# B&R Automation Studio project AsProject
Automation Studio 6.5.2.12; Starter Automation Studio project.; technology packages: mappConnect 6.1.0, mappView 6.6.0, OpcUaCs 6.5.0, OpcUaFx 6.6.0

## Configuration StarterConfig

CPU 5PC900.TS17-04, AutomationRuntime 6.5.1, Build 11.3.0

### Task classes (Cpu.sw)
```
Cyclic#1 (cycle 2000 us, tolerance 0 us):
  test <- test.prg
  TestTypes <- TestTypes.prg
  demo <- demo.prg
  demoGlobal <- demoGlobal.prg
  Page <- Page.prg
Binaries: udbdef, TCData, FWRules, mvLoader, mvDatApi, mvConfig, ashwd, ashwac, User, sysconf, asfw, arconfig, iomap, UaCsConfig, Config, BRRole, Role
Libraries: UaCore, ArSsl, FileIO, runtime
```

### Hardware
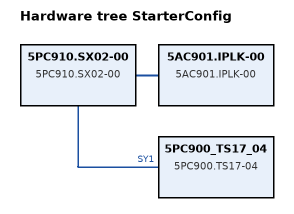
```
5AC901.IPLK-00 : 5AC901.IPLK-00 v2.1.0.0  [SS -> 5PC910.SX02-00.SS2]
  Connector IF1:
    DNAConfiguration = manual
5PC900_TS17_04 : 5PC900.TS17-04 v2.2.0.0  [SY -> 5PC910.SX02-00.SY1]
  ConfigurationID = Starter_StarterConfig
  UserPartitionSize = 300
  Simulation = 1
  UserRamDevice = PCI.2.IPLK.SRAM
  UserRamSize = 500000
  RemMemDevice = PCI.2.IPLK.SRAM
  RemMemSize = 120000
  PermanentPvSize = 10000
  RemanentGlobalPvSize = 105000
  VolatileGlobalPvSize = 1000000
  TimerDeviceType = EPLX2X
  TimerDevice = 5AC901.IPLK-00.IF1
  IdleTaskClass = 3
  TaskClassIdleTime = 8000
  Cyclic1Duration = 2000
  Cyclic1Tolerance = 0
  Cyclic2Duration = 10000
  Cyclic3Duration = 20000
  Cyclic3Tolerance = 40000
  FileDevice1
  FileDeviceName1 = USER
  FileDevicePath1 = USER_PATH
  TimeZone = 25
  ActivateFtpServer = 1
  FtpUser1
  FtpUsername1 = dev
  FtpUserPassword1 = NYwXHzz4INzZvtlFBMOTmjZqrH4JRkY3Uye1yrmlNSg=  // dev
  FtpUserSalt1 = s9/ksXy4
  FTPAccessRight1 = 0
  FTPdevice1 = ALL
  ActivateWebServer = 1
  ActivateSdm = 1
  SdmColor = colorRGB
  ActivateHypervisor = 1
5PC910.SX02-00 : 5PC910.SX02-00 v2.1.2.0
  Connector IF1:
    AssignedOperatingSystem = ARemb
  Connector IF3:
    AssignedOperatingSystem = ARemb
    ActivateDevice = 1
  Connector IF4:
    AssignedOperatingSystem = ARemb
    ActivateDevice = 1
  Connector IF10:
    OperatingSystem = ARemb
    ActivateDevice = 1
  Connector IF5:
    AssignedOperatingSystem = ARemb
  Connector IF6:
    AssignedOperatingSystem = ARemb
  Connector IF7:
    AssignedOperatingSystem = ARemb
  Connector IF8:
    AssignedOperatingSystem = ARemb
  Connector IF9:
    AssignedOperatingSystem = ARemb
```

### BRRole.brrole - 5PC900_TS17_04/AccessAndSecurity/UserRoleSystem/BRRole.brrole
```
Element BR_Anonymous (Type=BRRole)
Element BR_Engineer (Type=BRRole)
Element BR_Observer (Type=BRRole)
Element BR_SafetyAdmin (Type=BRRole)
Element BR_SecurityAdmin (Type=BRRole)
```

- Physical/StarterConfig/5PC900_TS17_04/IoMap.iom: same as Physical/StarterConfig/5PC900_TS17_04/Cpu.per
- Physical/StarterConfig/5PC900_TS17_04/PvMap.vvm: same as Physical/StarterConfig/5PC900_TS17_04/Cpu.per
### Config.mappconnect - 5PC900_TS17_04/mappConnect/Config.mappconnect
```
Element mapp Connect Configuration (Type=mappconnect)
  WebServerProtocol:
    WebServerPortSsl = 8443
    Interface = All
    SSLConfiguration = 
  WebServerEndpointConfiguration:
    Endpoint[1]:
      Endpoint = /Index.html
      Roles
    Endpoint[2]:
      Endpoint = /api/*
      Roles
    Endpoint[3]:
      Endpoint = /*
      Roles
  OpcUaServerWhitelist:
    OpcUaServer[1]:
      Url = opc.tcp://127.0.0.1:4840
```

## Logical view

### Global.var - Global variables
```iecst
VAR
	gRequestedMode : TestEnum;
	gActiveMode : TestEnum;
	testarray : TestArrays;
	gSimple : REAL;
	gtest : TestStruct;
END_VAR
```

### Types.typ - Local data types
```iecst
TYPE
	TestStruct : {REDUND_UNREPLICABLE} 	STRUCT
		command : {REDUND_UNREPLICABLE} BOOL;
		slider : {REDUND_UNREPLICABLE} REAL;
		random : {REDUND_UNREPLICABLE} REAL;
		_int : {REDUND_UNREPLICABLE} INT;
		_bool : {REDUND_UNREPLICABLE} BOOL;
		_real : {REDUND_UNREPLICABLE} REAL;
		_lreal : {REDUND_UNREPLICABLE} LREAL;
		struct2 : {REDUND_UNREPLICABLE} TestStruct1;
		struct3 : {REDUND_UNREPLICABLE} TestStruct1;
		struct1 : {REDUND_UNREPLICABLE} TestStruct1;
		myvalue : {REDUND_UNREPLICABLE} TestStruct3;
	END_STRUCT;
	TestStruct1 : {REDUND_UNREPLICABLE} 	STRUCT
		struct1 : {REDUND_UNREPLICABLE} TestStruct2;
		struct2 : {REDUND_UNREPLICABLE} TestStruct2;
	END_STRUCT;
	TestStruct2 : {REDUND_UNREPLICABLE} 	STRUCT
		member : {REDUND_UNREPLICABLE} BOOL;
		member1 : {REDUND_UNREPLICABLE} INT;
		member2 : {REDUND_UNREPLICABLE} DINT;
		member3 : {REDUND_UNREPLICABLE} STRING[80];
	END_STRUCT;
	TestStruct3 : {REDUND_UNREPLICABLE} 	STRUCT
		x : {REDUND_UNREPLICABLE} REAL;
	END_STRUCT;
	TestSimpleArray : {REDUND_UNREPLICABLE} 	STRUCT
		reals : {REDUND_UNREPLICABLE} ARRAY[0..2]OF REAL;
		ints : {REDUND_UNREPLICABLE} ARRAY[0..2]OF INT;
	END_STRUCT;
	TestOffsetArray : {REDUND_UNREPLICABLE} 	STRUCT
		standard : {REDUND_UNREPLICABLE} ARRAY[0..2]OF REAL;
		offset : {REDUND_UNREPLICABLE} ARRAY[1..3]OF REAL;
	END_STRUCT;
	TestArrays : {REDUND_UNREPLICABLE} 	STRUCT
		testArrayStruct : {REDUND_UNREPLICABLE} ARRAY[0..3]OF TestStruct2;
		doubleArray : {REDUND_UNREPLICABLE} ARRAY[0..3,0..3]OF TestStruct2;
		doubleArrayOffset1 : {REDUND_UNREPLICABLE} ARRAY[1..3,1..3]OF TestStruct2;
		TestOffsetArray : {REDUND_UNREPLICABLE} TestOffsetArray;
		New_Member1 : {REDUND_UNREPLICABLE} TestSimpleArray;
		status : {REDUND_UNREPLICABLE} STRING[80];
		temperature : {REDUND_UNREPLICABLE} REAL;
	END_STRUCT;
	TestEnum :
		(
		Value1,
		Value2,
		Value3,
		Value4,
		Value5,
		Value6,
		Value7
		);
END_TYPE
```


### Program Logical/demo (IEC)

#### Main.st - Init, cyclic, exit code
```iecst
PROGRAM _INIT

	test;
	test_arrays;

END_PROGRAM

PROGRAM _CYCLIC

	// Increment cycle counter for pseudo-random behavior
	cycle_counter := cycle_counter + 1;
	IF cycle_counter > 1000000 THEN
		cycle_counter := 0;
	END_IF;

	// Create pseudo-random selector to choose between structures and manipulation types
	random_selector := cycle_counter MOD 10;  // 10 different cases

	CASE random_selector OF
		0, 1, 2, 3, 4: // Manipulate test structure (50% of the time)
			structure_size := SIZEOF(test);
			offset := DINT_TO_UDINT(cycle_counter MOD UDINT_TO_DINT(structure_size));

			// Alternate between different data sizes
			CASE (cycle_counter MOD 3) OF
				0: // Write single bytes
					byte_ref ACCESS ADR(test) + offset;
					byte_ref := DINT_TO_USINT(cycle_counter MOD 256);
				1: // Write words (2 bytes), ensure alignment
					offset := offset AND 16#FFFFFFFE; // Align to word boundary
					IF offset + 2 <= structure_size THEN
						word_ref ACCESS ADR(test) + offset;
						word_ref := DINT_TO_UINT(cycle_counter MOD 65536);
					END_IF;
				2: // Write double words (4 bytes), ensure alignment
					offset := offset AND 16#FFFFFFFC; // Align to dword boundary
					IF offset + 4 <= structure_size THEN
						dword_ref ACCESS ADR(test) + offset;
						dword_ref := DINT_TO_UDINT(cycle_counter MOD 4294967295);
					END_IF;
			END_CASE;

		5, 6, 7, 8, 9: // Manipulate test_arrays structure (50% of the time)
			structure_size := SIZEOF(test_arrays);
			offset := DINT_TO_UDINT((cycle_counter * 7) MOD UDINT_TO_DINT(structure_size));

			// Alternate between different data sizes
			CASE ((cycle_counter * 3) MOD 3) OF
				0: // Write single bytes
					byte_ref ACCESS ADR(test_arrays) + offset;
					byte_ref := DINT_TO_USINT((cycle_counter * 11) MOD 256);
				1: // Write words (2 bytes), ensure alignment
					offset := offset AND 16#FFFFFFFE; // Align to word boundary
					IF offset + 2 <= structure_size THEN
						word_ref ACCESS ADR(test_arrays) + offset;
						word_ref := DINT_TO_UINT((cycle_counter * 13) MOD 65536);
					END_IF;
				2: // Write double words (4 bytes), ensure alignment
					offset := offset AND 16#FFFFFFFC; // Align to dword boundary
					IF offset + 4 <= structure_size THEN
						dword_ref ACCESS ADR(test_arrays) + offset;
						dword_ref := DINT_TO_UDINT((cycle_counter * 17) MOD 4294967295);
					END_IF;
			END_CASE;
	END_CASE;

END_PROGRAM

PROGRAM _EXIT
	(* Insert code here *)

END_PROGRAM
```

#### Variables.var - Local variables
```iecst
VAR
	test_arrays : TestArrays;
	test : TestStruct;
	cycle_counter : DINT := 0;
	random_selector : DINT := 0;
	byte_ref : REFERENCE TO USINT;
	word_ref : REFERENCE TO UINT;
	dword_ref : REFERENCE TO UDINT;
	offset : UDINT;
	structure_size : UDINT;
END_VAR
```

### Program Logical/test (IEC)

#### Main.st - Init, cyclic, exit code
```iecst
PROGRAM _INIT

	test;
	test_arrays;
	gActiveMode;
	gRequestedMode;
END_PROGRAM

PROGRAM _CYCLIC

	updating := updating + 2;

END_PROGRAM

PROGRAM _EXIT
	(* Insert code here *)

END_PROGRAM
```

#### Variables.var - Local variables
```iecst
VAR
	updating : UDINT;
	test_arrays : TestArrays;
	test : TestStruct;
END_VAR
```

### Program Logical/demoGlobal (IEC)

#### Main.st - Init, cyclic, exit code
```iecst
PROGRAM _INIT
	gtest;
	testarray;
	gSimple;
END_PROGRAM

PROGRAM _CYCLIC
	(* Insert code here *)

END_PROGRAM

PROGRAM _EXIT
	(* Insert code here *)

END_PROGRAM
```

### Program Logical/Page (IEC)

#### Cyclic.st - Cyclic code
```iecst
PROGRAM _CYCLIC
	(* Insert code here *)

END_PROGRAM
```

#### Init.st - Init code
```iecst
PROGRAM _INIT
	(* Insert code here *)

END_PROGRAM
```

#### Exit.st - Exit code
```iecst
PROGRAM _EXIT
	(* Insert code here *)

END_PROGRAM
```

#### Types.typ - Local data types
```iecst
TYPE
	myVar_typ : 	STRUCT
		in : myVar_in_typ;
		out : myVar_out_typ;
	END_STRUCT;
	myVar_in_typ : 	STRUCT
		command : USINT;
	END_STRUCT;
	myVar_out_typ : 	STRUCT
		state : USINT;
	END_STRUCT;
END_TYPE
```

#### Variables.var - Local variables
```iecst
VAR
	MyVar : myVar_typ;
END_VAR
```

### Package Logical/mappConnect/wwwRoot - wwwRoot

### TestTypes.typ
```iecst
(*
================================================================================
OPC UA Type Coverage Test Type Definitions
================================================================================
Structure type definitions for comprehensive OPC UA type testing

SETUP INSTRUCTIONS:
1. Import this .typ file into your PLC project data types
2. Import TestTypes.var for variable declarations
3. Map variables to OPC UA namespace 5

These structures are designed to test:
- Mixed primitive types in structures
- Nested structures
- Arrays of structures
- Deep field access (struct.member.submember)
================================================================================
*)

TYPE
    (* ====================================================================== *)
    (* Inner Structure for Nested Testing                                    *)
    (* ====================================================================== *)
    InnerStruct : STRUCT
        value : INT := 0;           (* Nested integer value *)
        enabled : BOOL := FALSE;    (* Nested boolean flag *)
    END_STRUCT;

    (* ====================================================================== *)
    (* Outer Structure Containing Inner Structure                            *)
    (* Tests: nestedStruct.inner.value access pattern                        *)
    (* ====================================================================== *)
    OuterStruct : STRUCT
        id : DINT := 0;             (* Outer level ID *)
        name : STRING[40] := '';    (* Outer level name *)
        inner : InnerStruct;        (* Nested structure *)
    END_STRUCT;

    (* ====================================================================== *)
    (* Structure with All Primitive Types                                    *)
    (* Tests: Reading/writing structures with mixed data types               *)
    (* Also tests individual member access: allTypesStruct.intVal, etc.      *)
    (* ====================================================================== *)
    AllTypesStruct : STRUCT
        intVal : INT := 0;          (* Signed 16-bit integer *)
        floatVal : REAL := 0.0;     (* 32-bit floating point *)
        boolVal : BOOL := FALSE;    (* Boolean value *)
        strVal : STRING[40] := '';  (* String value *)
        uint16Val : UINT := 0;      (* Unsigned 16-bit integer *)
        sint8Val : SINT := 0;       (* Signed 8-bit integer *)
        lrealVal : LREAL := 0.0;    (* 64-bit floating point *)
    END_STRUCT;

END_TYPE
```

### Program Logical/TestTypes (IEC)

#### Cyclic.st - Cyclic code
```iecst
PROGRAM _CYCLIC
	int8;// : SINT := 0; (* -128 to 127 *)
	int16;// : INT := 0; (* -32768 to 32767 *)
	int32;// : DINT := 0; (* -2147483648 to 2147483647 *)
	uint8;// : USINT := 0; (* 0 to 255 - also known as BYTE *)
	uint16;// : UINT := 0; (* 0 to 65535 - also known as WORD *)
	uint32;// : UDINT := 0; (* 0 to 4294967295 - also known as DWORD *)
	float32;// : REAL := 0.0; (* 32-bit single precision *)
	float64;// : LREAL := 0.0; (* 64-bit double precision *) (* ====================================================================== *) (* Boolean Type                                                           *)
	bool;// : BOOL := FALSE; (* TRUE or FALSE *) (* ====================================================================== *) (* String Types                                                           *)
	str;// : STRING[80] := ''; (* Standard ASCII string, max 80 chars *)
	wstr;// : WSTRING[80] := ""; (* Wide string (Unicode), max 80 chars *) (* ====================================================================== *) (* Date and Time Types                                                    *)
	dt;// : DATE_AND_TIME; (* Date and time combined *)
	tod;// : TIME_OF_DAY; (* Time of day only *)
	dateonly;// : DATE; (* Date only *) (* ====================================================================== *) (* Array Types - Primitives                                              *)
	intArr;// : ARRAY[0..9] OF INT := [10(0)]; (* Array of 10 integers *)
	realArr;// : ARRAY[0..9] OF REAL := [10(0.0)]; (* Array of 10 floats *)
	boolArr;// : ARRAY[0..9] OF BOOL := [10(FALSE)]; (* Array of 10 booleans *)
	strArr;// : ARRAY[0..4] OF STRING[40] := [5('')]; (* Array of 5 strings *) (* ====================================================================== *) (* Structure with All Primitive Types                                    *)
	allTypesStruct;// : AllTypesStruct := (intVal:=0,floatVal:=0.0,boolVal:=FALSE,strVal:='',uint16Val:=0,sint8Val:=0,lrealVal:=0.0); (* ====================================================================== *) (* Nested Structures                                                      *) (* Tests structure containing another structure                          *)
	nestedStruct;// : OuterStruct := (id:=0,name:='',inner:=(value:=0,enabled:=FALSE)); (* ====================================================================== *) (* Array of Structures                                                    *) (* Tests complex data type arrays                                        *)
	structArr;// : ARRAY[0..4] OF AllTypesStruct := [5((intVal:=0,floatVal:=0.0,boolVal:=FALSE,strVal:='',uint16Val:=0,sint8Val:=0,lrealVal:=0.0))];

END_PROGRAM
```

#### Init.st - Init code
```iecst
PROGRAM _INIT
	(* Insert code here *)

END_PROGRAM
```

#### Exit.st - Exit code
```iecst
PROGRAM _EXIT
	(* Insert code here *)

END_PROGRAM
```

#### TestTypes.var
```iecst
(*
================================================================================
OPC UA Type Coverage Test Variables
================================================================================
Import this file into your PLC project to enable comprehensive type testing

SETUP INSTRUCTIONS:
1. Add this .var file to your global variable section
2. Import TestTypes.typ for structure definitions
3. Map these variables to OPC UA namespace 5
4. Enable OPC UA server with authentication (dev/dev)

USAGE:
- Run tests/integration/type-coverage.test.ts
- All OPC UA standard types are tested for read/write compliance
================================================================================
*)
(* ====================================================================== *)
(* Signed Integer Types - Full range testing                             *)
(* ====================================================================== *)
VAR
	int8 : SINT := 0; (* -128 to 127 *)
	int16 : INT := 0; (* -32768 to 32767 *)
	int32 : DINT := 0; (* -2147483648 to 2147483647 *)
	uint8 : USINT := 0; (* 0 to 255 - also known as BYTE *)
	uint16 : UINT := 0; (* 0 to 65535 - also known as WORD *)
	uint32 : UDINT := 0; (* 0 to 4294967295 - also known as DWORD *)
	float32 : REAL := 0.0; (* 32-bit single precision *)
	float64 : LREAL := 0.0; (* 64-bit double precision *) (* ====================================================================== *) (* Boolean Type                                                           *)
	bool : BOOL := FALSE; (* TRUE or FALSE *) (* ====================================================================== *) (* String Types                                                           *)
	str : STRING[80] := ''; (* Standard ASCII string, max 80 chars *)
	wstr : WSTRING[80] := ""; (* Wide string (Unicode), max 80 chars *) (* ====================================================================== *) (* Date and Time Types                                                    *)
	dt : DATE_AND_TIME; (* Date and time combined *)
	tod : TIME_OF_DAY; (* Time of day only *)
	dateonly : DATE; (* Date only *) (* ====================================================================== *) (* Array Types - Primitives                                              *)
	intArr : ARRAY[0..9] OF INT := [10(0)]; (* Array of 10 integers *)
	realArr : ARRAY[0..9] OF REAL := [10(0.0)]; (* Array of 10 floats *)
	boolArr : ARRAY[0..9] OF BOOL := [10(FALSE)]; (* Array of 10 booleans *)
	strArr : ARRAY[0..4] OF STRING[40] := [5('')]; (* Array of 5 strings *) (* ====================================================================== *) (* Structure with All Primitive Types                                    *)
	allTypesStruct : AllTypesStruct := (intVal:=0,floatVal:=0.0,boolVal:=FALSE,strVal:='',uint16Val:=0,sint8Val:=0,lrealVal:=0.0); (* ====================================================================== *) (* Nested Structures                                                      *) (* Tests structure containing another structure                          *)
	nestedStruct : OuterStruct := (id:=0,name:='',inner:=(value:=0,enabled:=FALSE)); (* ====================================================================== *) (* Array of Structures                                                    *) (* Tests complex data type arrays                                        *)
	structArr : ARRAY[0..4] OF AllTypesStruct := [5((intVal:=0,floatVal:=0.0,boolVal:=FALSE,strVal:='',uint16Val:=0,sint8Val:=0,lrealVal:=0.0))];
END_VAR
```
